FUNCTION_BLOCK CAerationLogicBasic2 (* Basic Function Block Type *)
  (* Standard: 61499-2 *)
  (* Version 4.0, 9/29/2026, Schneider Electric, Rev4 - Limite 3, continuidade (transfere sem desligar) e alocacao so por rota passavel *)
  PACKAGE SE.Nereda;
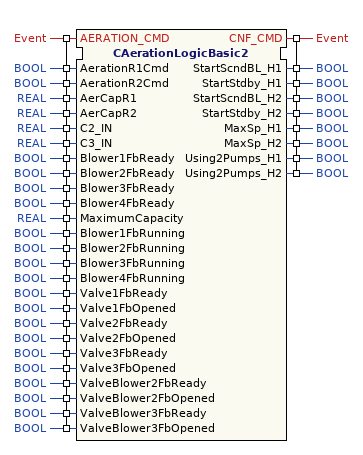
  EVENT_INPUT
    AERATION_CMD WITH AerationR1Cmd, AerationR2Cmd, AerCapR1, AerCapR2, C2_IN, C3_IN, Blower1FbReady, Blower2FbReady, Blower3FbReady, Blower4FbReady, MaximumCapacity, Blower1FbRunning, Blower2FbRunning, Blower3FbRunning, Blower4FbRunning, Valve1FbReady, Valve1FbOpened, Valve2FbReady, Valve2FbOpened, Valve3FbReady, Valve3FbOpened, ValveBlower2FbReady, ValveBlower2FbOpened, ValveBlower3FbReady, ValveBlower3FbOpened;
  END_EVENT
  EVENT_OUTPUT
    CNF_CMD WITH StartScndBL_H1, StartStdby_H1, StartScndBL_H2, StartStdby_H2, MaxSp_H1, MaxSp_H2, Using2Pumps_H1, Using2Pumps_H2;
  END_EVENT
  VAR_INPUT
    AerationR1Cmd : BOOL;
    AerationR2Cmd : BOOL;
    AerCapR1 : REAL;
    AerCapR2 : REAL;
    C2_IN : REAL;
    C3_IN : REAL;
    Blower1FbReady : BOOL;
    Blower2FbReady : BOOL;
    Blower3FbReady : BOOL;
    Blower4FbReady : BOOL;
    MaximumCapacity : REAL;
    Blower1FbRunning : BOOL;
    Blower2FbRunning : BOOL;
    Blower3FbRunning : BOOL;
    Blower4FbRunning : BOOL;
    Valve1FbReady : BOOL;
    Valve1FbOpened : BOOL;
    Valve2FbReady : BOOL;
    Valve2FbOpened : BOOL;
    Valve3FbReady : BOOL;
    Valve3FbOpened : BOOL;
    ValveBlower2FbReady : BOOL;
    ValveBlower2FbOpened : BOOL;
    ValveBlower3FbReady : BOOL;
    ValveBlower3FbOpened : BOOL;
  END_VAR
  VAR_OUTPUT
    StartScndBL_H1 : BOOL;
    StartStdby_H1 : BOOL;
    StartScndBL_H2 : BOOL;
    StartStdby_H2 : BOOL;
    MaxSp_H1 : BOOL;
    MaxSp_H2 : BOOL;
    Using2Pumps_H1 : BOOL;
    Using2Pumps_H2 : BOOL;
  END_VAR
  VAR
    Avail1 : BOOL;
    Avail2 : BOOL;
    Avail3 : BOOL;
    Avail4 : BOOL;
    Free2 : BOOL; (* Blower 2 livre para alocacao no ciclo *)
    Free3 : BOOL; (* Blower 3 livre para alocacao no ciclo *)
    Need2_H1 : BOOL := FALSE; (* Demanda R1 acima do SP (retido por histerese) *)
    Need2_H2 : BOOL := FALSE; (* Demanda R2 acima do SP (retido por histerese) *)
    NeedH1 : INT;
    NeedH2 : INT;
    CntH1 : INT;
    CntH2 : INT;
    H1_B2 : BOOL;
    H1_B3 : BOOL;
    H2_B3 : BOOL;
    H2_B2 : BOOL;
    HystPct : REAL := 5.0; (* Histerese de desligamento do 2o soprador em % de MaximumCapacity *)
    HystAbs : REAL;
    OutChanged : BOOL := FALSE;
    Initialized : BOOL := FALSE; (* Forca CNF_CMD no primeiro ciclo *)
    Last_StartScndBL_H1 : BOOL;
    Last_StartStdby_H1 : BOOL;
    Last_StartScndBL_H2 : BOOL;
    Last_StartStdby_H2 : BOOL;
    Last_MaxSp_H1 : BOOL;
    Last_MaxSp_H2 : BOOL;
    Last_Using2Pumps_H1 : BOOL;
    Last_Using2Pumps_H2 : BOOL;
    MaxBlowers : INT := 3; (* Maximo de sopradores ligados no total (B1..B4) *)
    SwapHystPct : REAL := 1.0; (* Histerese para trocar o reator que recebe o extra, em % de MaximumCapacity *)
    SwapHystAbs : REAL;
    Exc1 : REAL; (* AerCapR1 - MaximumCapacity *)
    Exc2 : REAL; (* AerCapR2 - MaximumCapacity *)
    ExtraPrio : INT := 0; (* Reator com prioridade no soprador extra: 0 nenhum, 1 R1, 2 R2 *)
    PassV1 : BOOL;
    PassV2 : BOOL;
    PassV3 : BOOL;
    PassVB2 : BOOL;
    PassVB3 : BOOL;
    Route2H1 : BOOL; (* B2 -> R1 passavel (VB2+V1) *)
    Route2H2 : BOOL; (* B2 -> R2 passavel (VB2+V2+V3) *)
    Route3H2 : BOOL; (* B3 -> R2 passavel (VB3+V3) *)
    Route3H1 : BOOL; (* B3 -> R1 passavel (VB3+V2+V1) *)
    PrevB2 : INT; (* Rota anterior do B2: 0 nenhuma, 1 R1, 2 R2 *)
    PrevB3 : INT; (* Rota anterior do B3 *)
    NewB2 : INT;
    NewB3 : INT;
    SwapRouteOk : BOOL;
  END_VAR
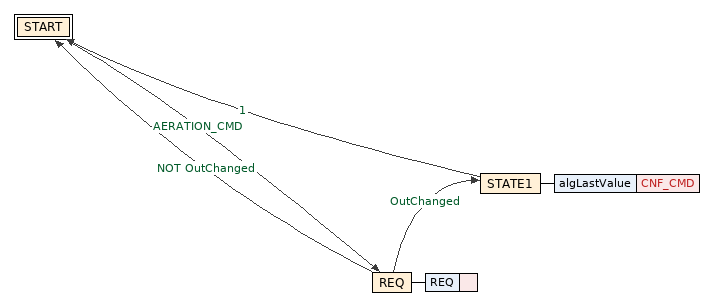
  EC_STATES
    START; (* Initial State *)
    REQ : REQ;
    STATE1 : algLastValue -> CNF_CMD;
  END_STATES
  EC_TRANSITIONS
    START TO REQ := AERATION_CMD;
    REQ TO STATE1 := OutChanged;
    STATE1 TO START := 1;
    REQ TO START := NOT OutChanged;
  END_TRANSITIONS
  ALGORITHM REQ IN ST:
;
(* ======================================================================== *)
(* CAerationLogicBasic2 - Rev4 (limite 3 + continuidade + rota passavel)    *)
(* Alocacao de sopradores por header                                        *)
(*   H1 (Reator 1): B1 fixo -> B2 (StartScndBL_H1) -> B3 (StartStdby_H1)     *)
(*   H2 (Reator 2): B4 fixo -> B3 (StartScndBL_H2) -> B2 (StartStdby_H2)     *)
(* Prioridades:                                                             *)
(*   1) Aeracao minima: 1 soprador em cada reator comandado                 *)
(*   2) Capacidade: 2o soprador quando AerCapRx > MaximumCapacity           *)
(*   3) Em disputa pelo mesmo soprador compartilhado, o header "dono" vence *)
(*      (B2 -> H1, B3 -> H2). Aeracao minima SEMPRE vence capacidade extra. *)
(*   4) Sem 2o soprador disponivel e demanda acima do SP -> MaxSp_Hx        *)
(*   5) Maximo MaxBlowers (3) sopradores ligados no total; o extra vai para *)
(*      o reator com maior demanda acima do SP (com histerese de troca)     *)
(*   6) Continuidade: prefere transferir soprador rodando a parar/partir    *)
(*   7) So aloca por rota passavel (todas as valvulas Ready ou abertas).   *)
(*      Se a prioridade nao consegue receber, o extra vai para o outro.    *)
(* B1/B4 sao partidos fora deste FB (AerationRxCmd). Um soprador nunca e    *)
(* alocado aos dois headers ao mesmo tempo.                                 *)
(* ======================================================================== *)

(* ---------- 1. Disponibilidade ---------- *)
Avail1 := Blower1FbReady OR Blower1FbRunning;
Avail2 := Blower2FbReady OR Blower2FbRunning;
Avail3 := Blower3FbReady OR Blower3FbRunning;
Avail4 := Blower4FbReady OR Blower4FbRunning;

(* ---------- 2. Demanda por header (com histerese) ---------- *)
HystAbs := MaximumCapacity * HystPct / 100.0;

IF NOT AerationR1Cmd THEN
    Need2_H1 := FALSE;
ELSIF AerCapR1 > MaximumCapacity THEN
    Need2_H1 := TRUE;
ELSIF AerCapR1 <= (MaximumCapacity - HystAbs) THEN
    Need2_H1 := FALSE;
END_IF;

IF NOT AerationR2Cmd THEN
    Need2_H2 := FALSE;
ELSIF AerCapR2 > MaximumCapacity THEN
    Need2_H2 := TRUE;
ELSIF AerCapR2 <= (MaximumCapacity - HystAbs) THEN
    Need2_H2 := FALSE;
END_IF;

NeedH1 := 0;
IF AerationR1Cmd THEN
    IF Need2_H1 THEN NeedH1 := 2; ELSE NeedH1 := 1; END_IF;
END_IF;

NeedH2 := 0;
IF AerationR2Cmd THEN
    IF Need2_H2 THEN NeedH2 := 2; ELSE NeedH2 := 1; END_IF;
END_IF;

(* ---------- 2b. Rotas passaveis (ar consegue chegar ao reator) ---------- *)
(* Valvula passavel: Ready (pode abrir) ou ja aberta (ar ja passa).        *)
(* Rota com qualquer valvula sem Ready e nao aberta e descartada: o        *)
(* soprador vai para quem consegue recebe-lo.                              *)
PassV1  := Valve1FbReady OR Valve1FbOpened;
PassV2  := Valve2FbReady OR Valve2FbOpened;
PassV3  := Valve3FbReady OR Valve3FbOpened;
PassVB2 := ValveBlower2FbReady OR ValveBlower2FbOpened;
PassVB3 := ValveBlower3FbReady OR ValveBlower3FbOpened;

Route2H1 := PassVB2 AND PassV1;             (* B2 -> R1: VB2 + V1      *)
Route2H2 := PassVB2 AND PassV2 AND PassV3;  (* B2 -> R2: VB2 + V2 + V3 *)
Route3H2 := PassVB3 AND PassV3;             (* B3 -> R2: VB3 + V3      *)
Route3H1 := PassVB3 AND PassV2 AND PassV1;  (* B3 -> R1: VB3 + V2 + V1 *)

(* ---------- 3. Inicializa alocacao ---------- *)
H1_B2 := FALSE;
H1_B3 := FALSE;
H2_B3 := FALSE;
H2_B2 := FALSE;
Free2 := Avail2;
Free3 := Avail3;

CntH1 := 0;
IF AerationR1Cmd AND Avail1 THEN CntH1 := 1; END_IF;
CntH2 := 0;
IF AerationR2Cmd AND Avail4 THEN CntH2 := 1; END_IF;

(* ---------- 4. Etapa 1 - garantir aeracao minima ---------- *)
(* 4a. soprador compartilhado "dono" *)
IF (NeedH1 >= 1) AND (CntH1 = 0) AND Free2 AND Route2H1 THEN
    H1_B2 := TRUE; Free2 := FALSE; CntH1 := CntH1 + 1;
END_IF;
IF (NeedH2 >= 1) AND (CntH2 = 0) AND Free3 AND Route3H2 THEN
    H2_B3 := TRUE; Free3 := FALSE; CntH2 := CntH2 + 1;
END_IF;
(* 4b. soprador compartilhado cruzado (standby) *)
IF (NeedH1 >= 1) AND (CntH1 = 0) AND Free3 AND Route3H1 THEN
    H1_B3 := TRUE; Free3 := FALSE; CntH1 := CntH1 + 1;
END_IF;
IF (NeedH2 >= 1) AND (CntH2 = 0) AND Free2 AND Route2H2 THEN
    H2_B2 := TRUE; Free2 := FALSE; CntH2 := CntH2 + 1;
END_IF;

(* ---------- 5. Etapa 2 - capacidade acima do setpoint ---------- *)
(* Limite: no maximo MaxBlowers sopradores ligados no total (B1..B4).  *)
(* Quando os dois reatores pedem 2 e so cabe 1 extra, leva quem tiver  *)
(* maior excesso sobre MaximumCapacity. A prioridade so troca se o     *)
(* outro superar o atual em SwapHystPct % (evita ficar trocando B2/B3). *)
Exc1 := AerCapR1 - MaximumCapacity;
Exc2 := AerCapR2 - MaximumCapacity;
SwapHystAbs := MaximumCapacity * SwapHystPct / 100.0;

IF (NeedH1 = 2) AND (NeedH2 = 2) THEN
    IF ExtraPrio = 1 THEN
        IF Exc2 > (Exc1 + SwapHystAbs) THEN ExtraPrio := 2; END_IF;
    ELSIF ExtraPrio = 2 THEN
        IF Exc1 > (Exc2 + SwapHystAbs) THEN ExtraPrio := 1; END_IF;
    ELSIF Exc2 > Exc1 THEN
        ExtraPrio := 2;
    ELSE
        ExtraPrio := 1;
    END_IF;
ELSIF NeedH1 = 2 THEN
    ExtraPrio := 1;
ELSIF NeedH2 = 2 THEN
    ExtraPrio := 2;
ELSE
    ExtraPrio := 0;
END_IF;

IF ExtraPrio = 2 THEN
    (* H2 tem prioridade no soprador extra *)
    IF (CntH2 < NeedH2) AND ((CntH1 + CntH2) < MaxBlowers) AND Free3 AND Route3H2 THEN
        H2_B3 := TRUE; Free3 := FALSE; CntH2 := CntH2 + 1;
    END_IF;
    IF (CntH2 < NeedH2) AND ((CntH1 + CntH2) < MaxBlowers) AND Free2 AND Route2H2 THEN
        H2_B2 := TRUE; Free2 := FALSE; CntH2 := CntH2 + 1;
    END_IF;
    IF (CntH1 < NeedH1) AND ((CntH1 + CntH2) < MaxBlowers) AND Free2 AND Route2H1 THEN
        H1_B2 := TRUE; Free2 := FALSE; CntH1 := CntH1 + 1;
    END_IF;
    IF (CntH1 < NeedH1) AND ((CntH1 + CntH2) < MaxBlowers) AND Free3 AND Route3H1 THEN
        H1_B3 := TRUE; Free3 := FALSE; CntH1 := CntH1 + 1;
    END_IF;
ELSE
    (* H1 tem prioridade no soprador extra *)
    IF (CntH1 < NeedH1) AND ((CntH1 + CntH2) < MaxBlowers) AND Free2 AND Route2H1 THEN
        H1_B2 := TRUE; Free2 := FALSE; CntH1 := CntH1 + 1;
    END_IF;
    IF (CntH1 < NeedH1) AND ((CntH1 + CntH2) < MaxBlowers) AND Free3 AND Route3H1 THEN
        H1_B3 := TRUE; Free3 := FALSE; CntH1 := CntH1 + 1;
    END_IF;
    IF (CntH2 < NeedH2) AND ((CntH1 + CntH2) < MaxBlowers) AND Free3 AND Route3H2 THEN
        H2_B3 := TRUE; Free3 := FALSE; CntH2 := CntH2 + 1;
    END_IF;
    IF (CntH2 < NeedH2) AND ((CntH1 + CntH2) < MaxBlowers) AND Free2 AND Route2H2 THEN
        H2_B2 := TRUE; Free2 := FALSE; CntH2 := CntH2 + 1;
    END_IF;
END_IF;

(* ---------- 5c. Continuidade: transferir em vez de parar/partir ---------- *)
(* Se o resultado for "para um soprador que esta rodando e parte o outro",   *)
(* o que ja esta rodando assume a rota do outro (transferencia sem desligar). *)
(* Mesmos sopradores por reator: capacidade, limite e prioridade iguais.     *)
PrevB2 := 0;
IF Last_StartScndBL_H1 THEN PrevB2 := 1; ELSIF Last_StartStdby_H2 THEN PrevB2 := 2; END_IF;
PrevB3 := 0;
IF Last_StartScndBL_H2 THEN PrevB3 := 2; ELSIF Last_StartStdby_H1 THEN PrevB3 := 1; END_IF;

NewB2 := 0;
IF H1_B2 THEN NewB2 := 1; ELSIF H2_B2 THEN NewB2 := 2; END_IF;
NewB3 := 0;
IF H2_B3 THEN NewB3 := 2; ELSIF H1_B3 THEN NewB3 := 1; END_IF;

(* Rota que o soprador em operacao teria no reator que o outro ia assumir *)
IF NewB3 = 1 THEN SwapRouteOk := Route2H1; ELSE SwapRouteOk := Route2H2; END_IF;
IF (PrevB2 <> 0) AND (NewB2 = 0) AND Blower2FbRunning AND (PrevB3 = 0) AND (NewB3 <> 0) AND SwapRouteOk THEN
    NewB2 := NewB3;
    NewB3 := 0;
ELSE
    IF NewB2 = 1 THEN SwapRouteOk := Route3H1; ELSE SwapRouteOk := Route3H2; END_IF;
    IF (PrevB3 <> 0) AND (NewB3 = 0) AND Blower3FbRunning AND (PrevB2 = 0) AND (NewB2 <> 0) AND SwapRouteOk THEN
        NewB3 := NewB2;
        NewB2 := 0;
    END_IF;
END_IF;

H1_B2 := NewB2 = 1;
H2_B2 := NewB2 = 2;
H2_B3 := NewB3 = 2;
H1_B3 := NewB3 = 1;

(* ---------- 6. Saidas ---------- *)
StartScndBL_H1 := H1_B2;   (* Blower 2 -> Header 1 *)
StartStdby_H1  := H1_B3;   (* Blower 3 -> Header 1 *)
StartScndBL_H2 := H2_B3;   (* Blower 3 -> Header 2 *)
StartStdby_H2  := H2_B2;   (* Blower 2 -> Header 2 *)

Using2Pumps_H1 := CntH1 >= 2;
Using2Pumps_H2 := CntH2 >= 2;

(* Demanda acima do SP sem 2o soprador: roda o(s) disponivel(is) no maximo *)
MaxSp_H1 := AerationR1Cmd AND (CntH1 >= 1) AND (CntH1 < NeedH1);
MaxSp_H2 := AerationR2Cmd AND (CntH2 >= 1) AND (CntH2 < NeedH2);

(* ---------- 7. Deteccao de mudanca (dispara CNF_CMD) ---------- *)
OutChanged := (NOT Initialized) OR
              (Last_StartScndBL_H1 <> StartScndBL_H1) OR
              (Last_StartStdby_H1 <> StartStdby_H1) OR
              (Last_StartScndBL_H2 <> StartScndBL_H2) OR
              (Last_StartStdby_H2 <> StartStdby_H2) OR
              (Last_MaxSp_H1 <> MaxSp_H1) OR
              (Last_MaxSp_H2 <> MaxSp_H2) OR
              (Last_Using2Pumps_H1 <> Using2Pumps_H1) OR
              (Last_Using2Pumps_H2 <> Using2Pumps_H2);
  END_ALGORITHM
  ALGORITHM algLastValue IN ST:
;
Last_StartScndBL_H1 := StartScndBL_H1;
Last_StartStdby_H1 := StartStdby_H1;
Last_StartScndBL_H2 := StartScndBL_H2;
Last_StartStdby_H2 := StartStdby_H2;
Last_MaxSp_H1 := MaxSp_H1;
Last_MaxSp_H2 := MaxSp_H2;
Last_Using2Pumps_H1 := Using2Pumps_H1;
Last_Using2Pumps_H2 := Using2Pumps_H2;
Initialized := TRUE;
  END_ALGORITHM
END_FUNCTION_BLOCK
